# EPICS substitutions: apps/plcApp/Db/solenoid_quench.substitutions
#
# solenoid_quench.substitions - Fast DAQ Quench Detection
#
# Author: Wesley Moore (wmoore@jlab.org)
# Date:   Nov 2016
#

file "db/torus_ai_generic.db" {
    pattern{ PLCID, P, R, TAG, EGU, PREC, DESC }
    { PLC_SOL, B_SOL:, QD:, VT1_DAQ,  V, 5, "raw input" }
    { PLC_SOL, B_SOL:, QD:, VT2_DAQ,  V, 5, "raw input" }
    { PLC_SOL, B_SOL:, QD:, VT3_DAQ,  V, 5, "raw input" }
    { PLC_SOL, B_SOL:, QD:, VT4_DAQ,  V, 5, "raw input" }
    { PLC_SOL, B_SOL:, QD:, VT5_DAQ,  V, 5, "raw input" }
    { PLC_SOL, B_SOL:, QD:, VT6_DAQ,  V, 5, "raw input" }
    { PLC_SOL, B_SOL:, QD:, VT7_DAQ,  V, 5, "raw input" }
    { PLC_SOL, B_SOL:, QD:, VT8_DAQ,  V, 5, "raw input" }
    { PLC_SOL, B_SOL:, QD:, VT9_DAQ,  V, 5, "raw input" }
    { PLC_SOL, B_SOL:, QD:, VT10_DAQ, V, 5, "raw input" }
    { PLC_SOL, B_SOL:, QD:, VT11_DAQ, V, 5, "raw input" }
    { PLC_SOL, B_SOL:, QD:, VT12_DAQ, V, 5, "raw input" }
    { PLC_SOL, B_SOL:, QD:, VT13_DAQ, V, 5, "raw input" }
    { PLC_SOL, B_SOL:, QD:, VT14_DAQ, V, 5, "raw input" }
    { PLC_SOL, B_SOL:, QD:, VT15_DAQ, V, 5, "raw input" }
    { PLC_SOL, B_SOL:, QD:, VT16_DAQ, V, 5, "raw input" }
    { PLC_SOL, B_SOL:, QD:, VT17_DAQ, V, 5, "raw input" }
    { PLC_SOL, B_SOL:, QD:, VT18_DAQ, V, 5, "raw input" }
    { PLC_SOL, B_SOL:, QD:, VT19_DAQ, V, 5, "raw input" }
    { PLC_SOL, B_SOL:, QD:, VT20_DAQ, V, 5, "raw input" }
    { PLC_SOL, B_SOL:, QD:, VT21_DAQ, V, 5, "raw input" }
    #
    { PLC_SOL, B_SOL:, QD:, V1,  V, 5, "plc calc" }
    { PLC_SOL, B_SOL:, QD:, V2,  V, 5, "plc calc" }
    { PLC_SOL, B_SOL:, QD:, V3,  V, 5, "plc calc" }
    { PLC_SOL, B_SOL:, QD:, V4,  V, 5, "plc calc" }
    { PLC_SOL, B_SOL:, QD:, V5,  V, 5, "plc calc" }
    { PLC_SOL, B_SOL:, QD:, V6,  V, 5, "plc calc" }
    { PLC_SOL, B_SOL:, QD:, V7,  V, 5, "plc calc" }
    { PLC_SOL, B_SOL:, QD:, V8,  V, 5, "plc calc" }
    { PLC_SOL, B_SOL:, QD:, V9,  V, 5, "plc calc" }
    { PLC_SOL, B_SOL:, QD:, V10, V, 5, "plc calc" }
    { PLC_SOL, B_SOL:, QD:, V11, V, 5, "plc calc" }
    { PLC_SOL, B_SOL:, QD:, V12, V, 5, "plc calc" }
    { PLC_SOL, B_SOL:, QD:, V13, V, 5, "plc calc" }
    { PLC_SOL, B_SOL:, QD:, V14, V, 5, "plc calc" }
    { PLC_SOL, B_SOL:, QD:, V15, V, 5, "plc calc" }
    #
    { PLC_SOL, B_SOL:, QD:, COMP1,  V, 5, "V1-V2" }
    { PLC_SOL, B_SOL:, QD:, COMP2,  V, 5, "V3-V4" }
    { PLC_SOL, B_SOL:, QD:, COMP3,  V, 5, "V5" }
    { PLC_SOL, B_SOL:, QD:, COMP4,  V, 5, "V6" }
    { PLC_SOL, B_SOL:, QD:, COMP5,  V, 5, "V7" }
    { PLC_SOL, B_SOL:, QD:, COMP6,  V, 5, "V8" }
    { PLC_SOL, B_SOL:, QD:, COMP7,  V, 5, "V9" }
    { PLC_SOL, B_SOL:, QD:, COMP8,  V, 5, "V10" }
    { PLC_SOL, B_SOL:, QD:, COMP9,  V, 5, "V11-V12" }
    { PLC_SOL, B_SOL:, QD:, COMP10, V, 5, "V13-V14" }
}

file "db/torus_bi_renamed.db" {
    pattern{ PLCID, P, R, PV, TAG, DESC }
    { PLC_SOL, B_SOL:, QD:, 1_CH1_LWR, QD1_Ch1_L, "QD1:CH1 Lower" }
    { PLC_SOL, B_SOL:, QD:, 1_CH1_UPR, QD1_Ch1_U, "QD1:CH1 Upper" }
    { PLC_SOL, B_SOL:, QD:, 1_CH2_LWR, QD1_Ch2_L, "QD1:CH2 Lower" }
    { PLC_SOL, B_SOL:, QD:, 1_CH2_UPR, QD1_Ch2_U, "QD1:CH2 Upper" }
    { PLC_SOL, B_SOL:, QD:, 1_CH3_LWR, QD1_Ch3_L, "QD1:CH3 Lower" }
    { PLC_SOL, B_SOL:, QD:, 1_CH3_UPR, QD1_Ch3_U, "QD1:CH3 Upper" }
    { PLC_SOL, B_SOL:, QD:, 1_CH4_LWR, QD1_Ch4_L, "QD1:CH4 Lower" }
    { PLC_SOL, B_SOL:, QD:, 1_CH4_UPR, QD1_Ch4_U, "QD1:CH4 Upper" }
    { PLC_SOL, B_SOL:, QD:, 2_CH1_LWR, QD2_Ch1_L, "QD2:CH1 Lower" }
    { PLC_SOL, B_SOL:, QD:, 2_CH1_UPR, QD2_Ch1_U, "QD2:CH1 Upper" }
    { PLC_SOL, B_SOL:, QD:, 2_CH2_LWR, QD2_Ch2_L, "QD2:CH2 Lower" }
    { PLC_SOL, B_SOL:, QD:, 2_CH2_UPR, QD2_Ch2_U, "QD2:CH2 Upper" }
    { PLC_SOL, B_SOL:, QD:, 2_CH3_LWR, QD2_Ch3_L, "QD2:CH3 Lower" }
    { PLC_SOL, B_SOL:, QD:, 2_CH3_UPR, QD2_Ch3_U, "QD2:CH3 Upper" }
    { PLC_SOL, B_SOL:, QD:, 2_CH4_LWR, QD2_Ch4_L, "QD2:CH4 Lower" }
    { PLC_SOL, B_SOL:, QD:, 2_CH4_UPR, QD2_Ch4_U, "QD2:CH4 Upper" }
}

file "db/torus_bo_renamed.db" {
    pattern{ PLCID, P, R, PV, TAG, DESC }
    { PLC_SOL, B_SOL:, QD:, MPS_Reset, MPS_Reset, "Hard Reset QD Power Supply" }
}

################################
# from cRIO
# - VT#_AVG
# - VT#_MAX
# - VT#_MIN
################################
file "db/solenoid_qd.db" {
    pattern{ P, R, VT, EGU, PREC, SCAN }
    { B_SOL:, QD:, VT1,  V, 5, "1 second" }
    { B_SOL:, QD:, VT2,  V, 5, "1 second" }
    { B_SOL:, QD:, VT3,  V, 5, "1 second" }
    { B_SOL:, QD:, VT4,  V, 5, "1 second" }
    { B_SOL:, QD:, VT5,  V, 5, "1 second" }
    { B_SOL:, QD:, VT6,  V, 5, "1 second" }
    { B_SOL:, QD:, VT7,  V, 5, "1 second" }
    { B_SOL:, QD:, VT8,  V, 5, "1 second" }
    { B_SOL:, QD:, VT9,  V, 5, "1 second" }
    { B_SOL:, QD:, VT10, V, 5, "1 second" }
    { B_SOL:, QD:, VT11, V, 5, "1 second" }
    { B_SOL:, QD:, VT12, V, 5, "1 second" }
    { B_SOL:, QD:, VT13, V, 5, "1 second" }
    { B_SOL:, QD:, VT14, V, 5, "1 second" }
    { B_SOL:, QD:, VT15, V, 5, "1 second" }
    { B_SOL:, QD:, VT16, V, 5, "1 second" }
    { B_SOL:, QD:, VT17, V, 5, "1 second" }
    { B_SOL:, QD:, VT18, V, 5, "1 second" }
    { B_SOL:, QD:, VT19, V, 5, "1 second" }
    { B_SOL:, QD:, VT20, V, 5, "1 second" }
    { B_SOL:, QD:, VT21, V, 5, "1 second" }
    { B_SOL:, QD:, VT22, V, 5, "1 second" }
    { B_SOL:, QD:, VT23, V, 5, "1 second" }
    { B_SOL:, QD:, IDCCT1, A, 2, "1 second" }
}
